FUNCTION INTERNAL _EmitSignal
VAR_INPUT
	iSignal		: I_SignalNode;
	iArg		: I_Arg;
END_VAR
VAR
	i			: UDINT;
	nEnd		: UDINT;
END_VAR

IF iSignal.count = 0 THEN
	RETURN;
END_IF

nEnd := iSignal.id + iSignal.count - 1;
FOR i := iSignal.id TO nEnd DO
	_Broadcast.stEntry[i].iReceiver.Receive(iArg);
END_FOR

END_FUNCTION

(* stored: Version 1.1.0.1
   POU _EmitSignal: Id {05058019-6f21-4744-b331-59e12922221f}, SpecialFunc None *)
